// TwinCAT 3 PLC project PLC1
// ProgramVersion: 3.1.4026.19
// CompilerDefines: VISU_USEPROPERTYINFO
// libraries:
//   SimplePackML, * (Beckhoff Automation Poland)
//   Tc2_BABasic, * (Beckhoff Automation GmbH)
//   Tc2_Standard, * (Beckhoff Automation GmbH)
//   Tc2_System, * (Beckhoff Automation GmbH)
//   Tc2_Utilities, * (Beckhoff Automation GmbH)
//   Tc3_EventLogger, * (Beckhoff Automation GmbH)
//   Tc3_PackML_V2, * (Beckhoff Automation GmbH)
// project tree:
//   / ClassDiagram.TcCD (not stored), ClassDiagram_1.TcCD (not stored), GlobalTextList.TcGTLO, PlcTask.TcTTO, Visualization Manager.TcVMO (not stored)
//   POUs/Devices/ Relay.TcPOU, TemperatureSensor.TcPOU
//   POUs/ IncrementVar.TcPOU, IncrementVarInst.TcPOU, MAIN.TcPOU, TestFbInit.TcPOU, Testowy.TcPOU, Testowy2.TcPOU, Testowy3.TcPOU
//   POUs/PackML/ Machine.TcPOU, P_PackML.TcPOU
//   POUs/ZadanieOOP/Devices/ AnalogLedDisplay010.TcPOU, ButtonNO.TcPOU, ButtonNC.TcPOU, Potentiometer.TcPOU
//   POUs/ZadanieOOP/Interfaces/ I_Button.TcIO, I_LimitedStringBuilder.TcIO, I_StringBuilder.TcIO, StringBuilder.TcPOU
//   POUs/ZadanieOOP/Modules/ PumpController.TcPOU, PumpControllerWithLogger.TcPOU, SignalTower.TcPOU, VolumePump.TcPOU
//   POUs/ZadanieOOP/ P_Machine.TcPOU
//   POUs/Zadanie/ FB_JuicePumpSimulator.TcPOU, GVL_IO.TcGVL (excluded from build), P_JuicePump.TcPOU
//   VISUs/ Visualization.TcVIS
// real-time tasks:
//   TASK PlcTask: cycle T#10ms, priority 20, ADS port 350
// I/O:
//   DEVICE Device 1 (EtherCAT), AmsNetId 0.0.0.0.2.1
//     Term 1 (EK1200) [EK1200-5000 EtherCAT Power supply (2A E-Bus)]
//       Term 2 (EL1004) [EL1004 4Ch. Dig. Input 24V, 3ms]
//       Term 3 (EL2008)
//       Term 4 (EL3064) [EL3064 4Ch. Ana. Input 0-10V]
//       Term 5 (EL4008) [EL4008 8Ch. Ana. Output 0-10V, 12bit]
//       Term 6 (EL6910) [EL6910, TwinSAFE PLC]
//       Term 7 (EL6070) [EL6070 1Ch. Licensing-Terminal]
//       Term 8 (EL1904) [EL1904, 4 Ch. Safety Input 24V, TwinSAFE]
//         modules: Module 1 (FSOES)
//       Term 9 (EL2904) [EL2904, 4 Ch. Safety Output 24V, 0.5A, TwinSAFE]
//         modules: Module 1 (FSOES), Module 2 (DO)
//       Term 10 (EL1018) [EL1018 8Ch. Dig. Input 24V, 10µs]
//       Term 11 (EL3214-0090) [EL3214-0090 4Ch. Ana. Input PT100 (RTD), TwinSAFE SC]
//       Term 12 (EL2024) [EL2024 4Ch. Dig. Output 24V, 2A]
//       Term 13 (EK1110) [EK1110 EtherCAT extension]
// variable links:
//   (this object) <-> Device 1 (EtherCAT)/Term 1 (EK1200)/Term 11 (EL3214-0090)
//     PlcTask Inputs/MAIN.tempSensor.stInputData.MDP5001_320_Input/MDP5001_320_Status <-> RTD Inputs Channel 1/Status
//     PlcTask Inputs/MAIN.tempSensor.stInputData.MDP5001_320_Input/MDP5001_320_Value <-> RTD Inputs Channel 1/Value
//   (this object) <-> Device 1 (EtherCAT)/Term 1 (EK1200)/Term 2 (EL1004)
//     PlcTask Inputs/MAIN.testButton.bInput <-> Channel 2/Input
//     PlcTask Inputs/P_Machine.requestButton.bInput <-> Channel 3/Input
//     PlcTask Inputs/P_Machine.startButton.bInput <-> Channel 1/Input
//   (this object) <-> Device 1 (EtherCAT)/Term 1 (EK1200)/Term 3 (EL2008)
//     PlcTask Outputs/P_Machine.appleJuiceContoller.volumePump.pump.bOutput <-> Channel 3/Output
//     PlcTask Outputs/P_Machine.signalTower.lightGreen.bOutput <-> Channel 1/Output
//     PlcTask Outputs/P_Machine.signalTower.lightRed.bOutput <-> Channel 2/Output
//   (this object) <-> Device 1 (EtherCAT)/Term 1 (EK1200)/Term 4 (EL3064)
//     PlcTask Inputs/P_Machine.appleJuiceContoller.juiceSetter.nInput <-> AI Standard Channel 1/Value
//     PlcTask Inputs/P_Machine.orangeJuiceContoller.juiceSetter.nInput <-> AI Standard Channel 2/Value
//   (this object) <-> Device 1 (EtherCAT)/Term 1 (EK1200)/Term 5 (EL4008)
//     PlcTask Outputs/P_Machine.appleJuiceContoller.ledDisplay.nOutput <-> AO Outputs Channel 1/Analog output
//     PlcTask Outputs/P_Machine.orangeJuiceContoller.ledDisplay.nOutput <-> AO Outputs Channel 2/Analog output

CONFIGURATION PLC1
    RESOURCE PLC ON TwinCAT3
        TASK PlcTask(INTERVAL := T#10ms, PRIORITY := 20);
        PROGRAM MAIN WITH PlcTask : MAIN;
    END_RESOURCE
END_CONFIGURATION

// ---- POUs/Zadanie/GVL_IO.TcGVL
{attribute 'qualified_only'}
VAR_GLOBAL
	//wejscia
	bStart			AT%I*	: BOOL;
	bRequest		AT%I*	: BOOL;
	nJuiceSetter	AT%I*	: INT;
	//wyścia
	bLightSignal1	AT%Q*	: BOOL;
	bLightSignal2	AT%Q*	: BOOL;
	nLedDisplay		AT%Q*	: INT;
	bPump			AT%Q*	: BOOL;
END_VAR

// ---- POUs/ZadanieOOP/Interfaces/I_Button.TcIO
INTERFACE I_Button

PROPERTY IsPressed : BOOL
GET
END_GET
END_PROPERTY

PROPERTY IsReleased : BOOL
GET
END_GET
END_PROPERTY

PROPERTY RisingTrigger : BOOL
GET
END_GET
END_PROPERTY

END_INTERFACE

// ---- POUs/ZadanieOOP/Interfaces/I_LimitedStringBuilder.TcIO
INTERFACE I_LimitedStringBuilder

METHOD Append : I_StringBuilder
VAR_INPUT
	sText	: T_MaxString;
END_VAR
END_METHOD

METHOD Reset : I_LimitedStringBuilder
VAR_INPUT
END_VAR
END_METHOD

METHOD ToString : T_MaxString
VAR_INPUT
END_VAR
END_METHOD

END_INTERFACE

// ---- POUs/ZadanieOOP/Interfaces/I_StringBuilder.TcIO
INTERFACE I_StringBuilder

METHOD Append : I_StringBuilder
VAR_INPUT
	sText	: T_MaxString;
END_VAR
END_METHOD

METHOD Reset : I_LimitedStringBuilder
VAR_INPUT
END_VAR
END_METHOD

METHOD ToLowerCase : I_StringBuilder
VAR_INPUT
END_VAR
END_METHOD

METHOD ToString : T_MaxString
VAR_INPUT
END_VAR
END_METHOD

METHOD ToUpperCase : I_StringBuilder
VAR_INPUT
END_VAR
END_METHOD

END_INTERFACE

// ---- POUs/MAIN.TcPOU
PROGRAM MAIN
VAR
	nState		: UINT;
	motorRelay	: Relay;
	incVar		: IncrementVar;
	incVarInst	: IncrementVarInst;
	bTest		: BOOL;
	nVal1		: INT;
	nVal2		: INT;
	tempSensor	: TemperatureSensor;
	temperature	: REAL;
	offset		: REAL;
	
	testButton	: ButtonNC;
	testTrigger	: BOOL;
	
	testFbInit	: TestFbInit(wartosc := 7);
	
	pInt		: REFERENCE TO INT;
	nInt		: INT;
	nInt2		: INT;
	
	itfButton	: I_Button;
	buttonNo	: ButtonNO;
	buttonNc	: ButtonNC;
	bIsPressed	: BOOL;
	
	sTekst		: STRING;
	nNrAlarmu	: INT := 7;
	alarm 		: StringBuilder;
END_VAR

motorRelay.Cyclic();

CASE nState OF
	
	0:
		;
		
	10:
		IF motorRelay.SwitchOn() THEN
			nState := 0;
		END_IF
		
	20:
		IF motorRelay.SwitchOff() THEN
			nState := 0;
		END_IF
		
	30:
		IF motorRelay.Pulse(T#5S) THEN
			nState := 0;
		END_IF
		
	40:
		IF motorRelay.PulseAcyclic(T#5S) THEN
			nState := 0;
		END_IF
		
END_CASE

IF bTest THEN
	bTest := FALSE;
	nVal1 := incVar.Increment();
	nVal2 := incVarInst.Increment();
END_IF

tempSensor.OffsetInCelsius := -25;
temperature := tempSensor.InCelsius;
offset := tempSensor.OffsetInCelsius;

// P_JuicePump();
P_Machine();

IF testButton.RisingTrigger THEN
	testTrigger := TRUE;
END_IF

pInt REF= nInt2;

IF __ISVALIDREF(pInt) THEN
	nInt := pInt;
END_IF

itfButton := buttonNc;

IF itfButton <> 0 AND_THEN itfButton.IsPressed THEN
	bIsPressed := TRUE;
END_IF

// sTekst := alarm.Reset()
// 			.Append('Alarm nr: ')
// 			.Append(TO_STRING(nNrAlarmu))
// 			.Append(' Temperatura zbyt wysoka')
// 			.ToString();

P_PackML();

END_PROGRAM

// ---- POUs/Devices/Relay.TcPOU
FUNCTION_BLOCK Relay
VAR
	bOutput	AT%Q*	: BOOL;
	tonPulse		: TON;
	tonPulseAcyclic	: TON;
END_VAR

// tonPulseAcyclic();
// 
// IF tonPulseAcyclic.Q THEN
// 	SwitchOff();
// 	tonPulseAcyclic(IN := FALSE);
// END_IF

METHOD Cyclic
VAR_INPUT
END_VAR
tonPulseAcyclic();

IF tonPulseAcyclic.Q THEN
	SwitchOff();
	tonPulseAcyclic(IN := FALSE);
END_IF
END_METHOD

METHOD Pulse : BOOL
VAR_INPUT
	tPulseTime	: TIME;
END_VAR
tonPulse(IN := TRUE, PT:= tPulseTime);

IF NOT tonPulse.Q THEN
	SwitchOn();
ELSIF tonPulse.Q THEN
	SwitchOff();
	tonPulse(IN := FALSE);
	Pulse := TRUE;
END_IF
END_METHOD

METHOD PulseAcyclic : BOOL
VAR_INPUT
	tPulseTime	: TIME;
END_VAR
SwitchOn();
tonPulseAcyclic.IN := TRUE;
tonPulseAcyclic.PT := tPulseTime;

PulseAcyclic := TRUE;
END_METHOD

PROPERTY State : BOOL
GET
State := bOutput;
END_GET
END_PROPERTY

METHOD SwitchOff : BOOL
VAR_INPUT
END_VAR
bOutput := FALSE;

SwitchOff := TRUE;
END_METHOD

METHOD SwitchOn : BOOL
VAR_INPUT
END_VAR
bOutput := TRUE;

SwitchOn := TRUE;
END_METHOD

END_FUNCTION_BLOCK

// ---- POUs/IncrementVar.TcPOU
FUNCTION_BLOCK IncrementVar
VAR
END_VAR

METHOD Increment : INT
VAR
	nValue	: INT := 5;
END_VAR
nValue := nValue + 1;
Increment := nValue;
END_METHOD

END_FUNCTION_BLOCK

// ---- POUs/IncrementVarInst.TcPOU
FUNCTION_BLOCK IncrementVarInst
VAR
END_VAR

METHOD Increment : INT
VAR_INST
	nValue	: INT := 5;
END_VAR
nValue := nValue + 1;
Increment := nValue;
END_METHOD

END_FUNCTION_BLOCK

// ---- POUs/Devices/TemperatureSensor.TcPOU
FUNCTION_BLOCK TemperatureSensor
VAR
	stInputData			: MDP5001_320_A369A904;
	fOffsetInCelsius	: REAL;
END_VAR

{attribute 'monitoring' := 'call'}
PROPERTY Error : BOOL
GET
Error := stInputData.MDP5001_320_Input.MDP5001_320_Status.Error;
END_GET
END_PROPERTY

{attribute 'monitoring' := 'call'}
PROPERTY InCelsius : REAL
GET
InCelsius := (stInputData.MDP5001_320_Input.MDP5001_320_Value / 10.0) + fOffsetInCelsius;
END_GET
END_PROPERTY

{attribute 'monitoring' := 'call'}
PROPERTY InFarenheit : REAL
GET
InFarenheit := C_TO_F ( fX := InCelsius );
END_GET
END_PROPERTY

{attribute 'monitoring' := 'call'}
PROPERTY InKelvin : REAL
GET
InKelvin := C_TO_K ( fX := InCelsius );
END_GET
END_PROPERTY

{attribute 'monitoring' := 'call'}
PROPERTY InReaumur : REAL
GET
InReaumur := C_TO_R ( fX := InCelsius );
END_GET
END_PROPERTY

{attribute 'monitoring' := 'call'}
PROPERTY OffsetInCelsius : REAL
GET
OffsetInCelsius := fOffsetInCelsius;
END_GET
SET
fOffsetInCelsius := OffsetInCelsius;
END_SET
END_PROPERTY

{attribute 'monitoring' := 'call'}
PROPERTY Overrange : BOOL
GET
Overrange := stInputData.MDP5001_320_Input.MDP5001_320_Status.Overrange;
END_GET
END_PROPERTY

{attribute 'monitoring' := 'call'}
PROPERTY Underrange : BOOL
GET
Underrange := stInputData.MDP5001_320_Input.MDP5001_320_Status.Underrange;
END_GET
END_PROPERTY

END_FUNCTION_BLOCK

// ---- POUs/ZadanieOOP/Devices/ButtonNC.TcPOU
FUNCTION_BLOCK ButtonNC IMPLEMENTS I_Button
VAR
	bInput	AT%I*	: BOOL;
	rtInput			: R_TRIG;
END_VAR

PROPERTY IsPressed : BOOL
GET
IsPressed := NOT bInput;
END_GET
END_PROPERTY

PROPERTY IsReleased : BOOL
GET
IsReleased := NOT IsPressed;
END_GET
END_PROPERTY

PROPERTY RisingTrigger : BOOL
GET
rtInput(CLK := IsPressed);

RisingTrigger := rtInput.Q;
END_GET
END_PROPERTY

END_FUNCTION_BLOCK

// ---- POUs/TestFbInit.TcPOU
FUNCTION_BLOCK TestFbInit
VAR
	nValue	: INT := 5;
END_VAR

//FB_Init is always available implicitly and it is used primarily for initialization.
//The return value is not evaluated. For a specific influence, you can also declare the
//methods explicitly and provide additional code there with the standard initialization
//code. You can evaluate the return value.
METHOD FB_Init: BOOL
VAR_INPUT
    bInitRetains: BOOL; // TRUE: the retain variables are initialized (reset warm / reset cold)
    bInCopyCode: BOOL;  // TRUE: the instance will be copied to the copy code afterward (online change)
	wartosc		: INT;   
END_VAR
nValue := wartosc;
END_METHOD

END_FUNCTION_BLOCK

// ---- POUs/ZadanieOOP/Devices/ButtonNO.TcPOU
FUNCTION_BLOCK ButtonNO IMPLEMENTS I_Button
VAR
	bInput	AT%I*	: BOOL;
	rtInput			: R_TRIG;
END_VAR

PROPERTY IsPressed : BOOL
GET
IsPressed := bInput;
END_GET
END_PROPERTY

PROPERTY IsReleased : BOOL
GET
IsReleased := NOT IsPressed;
END_GET
END_PROPERTY

PROPERTY RisingTrigger : BOOL
GET
rtInput(CLK := IsPressed);

RisingTrigger := rtInput.Q;
END_GET
END_PROPERTY

END_FUNCTION_BLOCK

// ---- POUs/ZadanieOOP/Interfaces/StringBuilder.TcPOU
FUNCTION_BLOCK StringBuilder IMPLEMENTS I_LimitedStringBuilder, I_StringBuilder
VAR
	sBuiltString	: T_MaxString;
END_VAR

METHOD Append : I_StringBuilder
VAR_INPUT
	sText	: T_MaxString;
END_VAR
sBuiltString := CONCAT(sBuiltString, sText);

Append := THIS^;
END_METHOD

METHOD Reset : I_LimitedStringBuilder
sBuiltString := '';

Reset := THIS^;
END_METHOD

{warning 'Add method implementation '}
METHOD ToLowerCase : I_StringBuilder
END_METHOD

METHOD ToString : T_MaxString
ToString := sBuiltString;
END_METHOD

{warning 'Add method implementation '}
METHOD ToUpperCase : I_StringBuilder
END_METHOD

END_FUNCTION_BLOCK

// ---- POUs/ZadanieOOP/P_Machine.TcPOU
PROGRAM P_Machine
VAR
	startButton			: ButtonNO;
	requestButton		: ButtonNO;
	appleJuiceContoller	: PumpControllerWithLogger(requestButton, 0, 10_000);
	orangeJuiceContoller: PumpControllerWithLogger(requestButton, 0, 5_000);
	signalTower			: SignalTower;
END_VAR

appleJuiceContoller();
orangeJuiceContoller();

IF startButton.RisingTrigger THEN
	appleJuiceContoller.Enable();
	orangeJuiceContoller.Enable();
END_IF

IF appleJuiceContoller.IsDisabled THEN
	signalTower.SwitchOffGreen();
	signalTower.SwitchOffRed();
ELSIF appleJuiceContoller.IsEnabled THEN
	signalTower.SwitchOnGreen();
	signalTower.SwitchOffRed();
ELSIF appleJuiceContoller.IsPumping THEN
	signalTower.SwitchOnGreen();
	signalTower.SwitchOnRed();
ELSIF appleJuiceContoller.IsPumpingComplete THEN
	signalTower.SwitchOnGreen();
	signalTower.SwitchOffRed();
END_IF

END_PROGRAM

// ---- POUs/ZadanieOOP/Modules/PumpControllerWithLogger.TcPOU
FUNCTION_BLOCK PumpControllerWithLogger EXTENDS PumpController
VAR
	stringBuilder	: StringBuilder;
	logDataTrigger	: R_TRIG;
END_VAR
VAR_STAT
	nCycles			: UINT;
END_VAR

SUPER^();

LogToAds();

METHOD PRIVATE LogToAds : BOOL
VAR_INPUT
END_VAR
logDataTrigger(CLK := IsPumpingComplete);

IF logDataTrigger.Q THEN
	nCycles := nCycles + 1;
	
	stringBuilder.Reset()
		.Append('Lacznie wykonano: ')
		.Append(TO_STRING(nCycles))
		.Append(' cykli');
		
	ADSLOGSTR( msgCtrlMask := ADSLOG_MSGTYPE_LOG, msgFmtStr := stringBuilder.ToString(), strArg := '' );
END_IF
END_METHOD

END_FUNCTION_BLOCK

// ---- POUs/ZadanieOOP/Modules/PumpController.TcPOU
FUNCTION_BLOCK PumpController
VAR
	volumePump					: VolumePump;
	eState						: ( DISABLED, ENABLED, PUMPING, PUMPING_COMPLETE );
	requestButton				: I_Button;
	juiceSetter					: Potentiometer;
	ledDisplay					: AnalogLedDisplay010;
	fJuiceSetpointInMililiters	: LREAL;
	fMinSetRangeInMililiters	: LREAL;
	fMaxSetRangeInMililiters	: LREAL;
END_VAR

volumePump();

CASE eState OF
	
	DISABLED:
		;
		
	ENABLED:
		ledDisplay.SetValue(juiceSetter.ActualValue);
		IF requestButton.IsPressed THEN
			fJuiceSetpointInMililiters := F_Scale ( juiceSetter.ActualValue, 0, 32767, fMinSetRangeInMililiters, fMaxSetRangeInMililiters );
			eState := PUMPING;
		END_IF
		
	PUMPING:
		ledDisplay.SetValue( TO_INT (F_Scale ( fJuiceSetpointInMililiters - volumePump.PumpedJuiceInMililiters, fMinSetRangeInMililiters, fMaxSetRangeInMililiters, 0, 32767 ) ) );
		volumePump.Start();
		IF volumePump.PumpedJuiceInMililiters >= fJuiceSetpointInMililiters THEN
			volumePump.Reset();
			eState := PUMPING_COMPLETE;
		END_IF
		
	PUMPING_COMPLETE:
		;
		
END_CASE

METHOD Disable : BOOL
VAR_INPUT
END_VAR
eState := DISABLED;
END_METHOD

METHOD Enable : BOOL
VAR_INPUT
END_VAR
eState := ENABLED;
END_METHOD

//FB_Init is always available implicitly and it is used primarily for initialization.
//The return value is not evaluated. For a specific influence, you can also declare the
//methods explicitly and provide additional code there with the standard initialization
//code. You can evaluate the return value.
METHOD FB_Init: BOOL
VAR_INPUT
    bInitRetains: BOOL; // TRUE: the retain variables are initialized (reset warm / reset cold)
    bInCopyCode: BOOL;  // TRUE: the instance will be copied to the copy code afterward (online change)   
	requestButton				: I_Button;
	fMinSetRangeInMililiters	: LREAL;
	fMaxSetRangeInMililiters	: LREAL;
END_VAR
THIS^.requestButton := requestButton;
THIS^.fMinSetRangeInMililiters := LIMIT(0, fMinSetRangeInMililiters, 10_000);
THIS^.fMaxSetRangeInMililiters := LIMIT(0, fMaxSetRangeInMililiters, 10_000);
END_METHOD

PROPERTY IsDisabled : BOOL
GET
IsDisabled := eState = DISABLED;
END_GET
END_PROPERTY

PROPERTY IsEnabled : BOOL
GET
IsEnabled := eState = ENABLED;
END_GET
END_PROPERTY

PROPERTY IsPumping : BOOL
GET
IsPumping := eState = PUMPING;
END_GET
END_PROPERTY

PROPERTY IsPumpingComplete : BOOL
GET
IsPumpingComplete := eState = PUMPING_COMPLETE;
END_GET
END_PROPERTY

END_FUNCTION_BLOCK

// ---- POUs/ZadanieOOP/Modules/VolumePump.TcPOU
FUNCTION_BLOCK VolumePump
VAR
	pump						: Relay;
	eState						: ( RESET, START );
	fPumpedJuiceInMililiters	: REAL;
END_VAR

CASE eState OF
	
	RESET:
		pump.SwitchOff();
		fPumpedJuiceInMililiters := 0;
		
	START:
		pump.SwitchOn();
		fPumpedJuiceInMililiters := fPumpedJuiceInMililiters + 10;
		
END_CASE

PROPERTY IsPumping : BOOL
GET
IsPumping := pump.State;
END_GET
END_PROPERTY

PROPERTY PumpedJuiceInMililiters : REAL
GET
PumpedJuiceInMililiters := fPumpedJuiceInMililiters;
END_GET
END_PROPERTY

METHOD Reset : BOOL
VAR_INPUT
END_VAR
eState := RESET;
END_METHOD

METHOD Start : BOOL
VAR_INPUT
END_VAR
eState := START;
END_METHOD

END_FUNCTION_BLOCK

// ---- POUs/ZadanieOOP/Devices/Potentiometer.TcPOU
FUNCTION_BLOCK Potentiometer
VAR
	nInput	AT%I*	: INT;
END_VAR

PROPERTY ActualValue : INT
GET
ActualValue := nInput;
END_GET
END_PROPERTY

PROPERTY ActualValuePercent : LREAL
GET
ActualValuePercent := F_Scale ( nInput, 0, 32767, 0, 100 );
END_GET
END_PROPERTY

END_FUNCTION_BLOCK

// ---- POUs/ZadanieOOP/Devices/AnalogLedDisplay010.TcPOU
FUNCTION_BLOCK AnalogLedDisplay010
VAR
	nOutput	AT%Q*	: INT;
END_VAR

PROPERTY DisplayedValue : LREAL
GET
DisplayedValue := F_Scale ( nOutput, 0, 32767, 0, 10 );
END_GET
END_PROPERTY

METHOD SetValue : BOOL
VAR_INPUT
	nValue	: INT;
END_VAR
nOutput := nValue;

SetValue := TRUE;
END_METHOD

END_FUNCTION_BLOCK

// ---- POUs/ZadanieOOP/Modules/SignalTower.TcPOU
FUNCTION_BLOCK SignalTower
VAR
	lightGreen	: Relay;
	lightRed	: Relay;
END_VAR

PROPERTY GreenLightState : BOOL
GET
GreenLightState := lightGreen.State;
END_GET
END_PROPERTY

PROPERTY RedLightState : BOOL
GET
RedLightState := lightRed.State;
END_GET
END_PROPERTY

METHOD SwitchOffGreen : BOOL
VAR_INPUT
END_VAR
lightGreen.SwitchOff();
END_METHOD

METHOD SwitchOffRed : BOOL
VAR_INPUT
END_VAR
lightRed.SwitchOff();
END_METHOD

METHOD SwitchOnGreen : BOOL
VAR_INPUT
END_VAR
lightGreen.SwitchOn();
END_METHOD

METHOD SwitchOnRed : BOOL
VAR_INPUT
END_VAR
lightRed.SwitchOn();
END_METHOD

END_FUNCTION_BLOCK

// ---- POUs/PackML/P_PackML.TcPOU
PROGRAM P_PackML
VAR
	machine1	: Machine;
	eModeCommand: E_PMLProtectedUnitMode;
	eCommand	: E_PMLCommand;
END_VAR

machine1(
	eModeCommand	:= eModeCommand, 
	eCommand		:= eCommand, 
	eMode			=> , 
	eState			=> , 
	bUndefinedDone	=> , 
	bInvalidModeCommandOut=> , 
	bChangeIntoProduction=> );

END_PROGRAM

// ---- POUs/PackML/Machine.TcPOU
FUNCTION_BLOCK Machine EXTENDS FB_Generic
VAR
END_VAR

SUPER^();

METHOD M_Aborting
VAR_INST
	bTest	: BOOL;
END_VAR
IF bTest THEN
	bTest := FALSE;
	M_StateComplete();
END_IF
END_METHOD

METHOD M_Execute
VAR_INST
	bTest	: BOOL;
END_VAR
IF bTest THEN
	bTest := FALSE;
	M_StateComplete();
END_IF
END_METHOD

METHOD M_StateComplete
SUPER^.M_StateComplete();
END_METHOD

END_FUNCTION_BLOCK

// ---- POUs/Testowy.TcPOU
FUNCTION_BLOCK Testowy
VAR
END_VAR

END_FUNCTION_BLOCK

// ---- POUs/Testowy2.TcPOU
FUNCTION_BLOCK Testowy2
VAR
	bTest: BOOL;
END_VAR

END_FUNCTION_BLOCK

// ---- POUs/Testowy3.TcPOU
FUNCTION_BLOCK Testowy3
VAR
	bTest3: BOOL;
END_VAR

END_FUNCTION_BLOCK

// ---- POUs/Zadanie/FB_JuicePumpSimulator.TcPOU
FUNCTION_BLOCK FB_JuicePumpSimulator
VAR_INPUT
	bStart						: BOOL;
	bReset						: BOOL;
END_VAR
VAR_OUTPUT
	fPumpedJuiceInMililiters	: REAL;
END_VAR
VAR
	rtReset						: R_TRIG;
END_VAR

rtReset( CLK := bReset );
IF rtReset.Q THEN
	fPumpedJuiceInMililiters := 0;
END_IF

IF bStart THEN
	fPumpedJuiceInMililiters := fPumpedJuiceInMililiters + 10;		// 1kg / s
END_IF

END_FUNCTION_BLOCK

// ---- POUs/Zadanie/P_JuicePump.TcPOU
PROGRAM P_JuicePump
VAR
	eState						: ( DISABLED, ENABLED, PUMPING );
	fbPumpSimulator				: FB_JuicePumpSimulator;
	rtStartButton				: R_TRIG;
	ftStartButton				: F_TRIG;
	fJuiceSetpointInMililiters	: LREAL;
END_VAR

fbPumpSimulator( bStart := GVL_IO.bPump );
ftStartButton( CLK := GVL_IO.bStart );
IF ftStartButton.Q THEN
	fbPumpSimulator( bReset := TRUE );
	fbPumpSimulator( bReset := FALSE );
END_IF

CASE eState OF
	
	DISABLED:
		rtStartButton(CLK := GVL_IO.bStart);
		IF rtStartButton.Q THEN
			eState := ENABLED;
		END_IF
		
	ENABLED:
		GVL_IO.bLightSignal1 := TRUE;
		GVL_IO.nLedDisplay := GVL_IO.nJuiceSetter;
		IF GVL_IO.bRequest THEN
			fJuiceSetpointInMililiters := F_Scale ( GVL_IO.nJuiceSetter, 0, 32767, 0, 10_000 );
			eState := PUMPING;
		END_IF
		
	PUMPING:
		GVL_IO.nLedDisplay := TO_INT (F_Scale ( fJuiceSetpointInMililiters - fbPumpSimulator.fPumpedJuiceInMililiters, 0, 10_000, 0, 32767 ) );
		GVL_IO.bLightSignal2 := TRUE;
		GVL_IO.bPump := TRUE;
		IF fbPumpSimulator.fPumpedJuiceInMililiters >= fJuiceSetpointInMililiters THEN
			GVL_IO.bLightSignal1 := FALSE;
			GVL_IO.bLightSignal2 := FALSE;
			GVL_IO.bPump := FALSE;
			eState := DISABLED;
		END_IF
		
END_CASE

END_PROGRAM

// ---- VISUs/Visualization.TcVIS
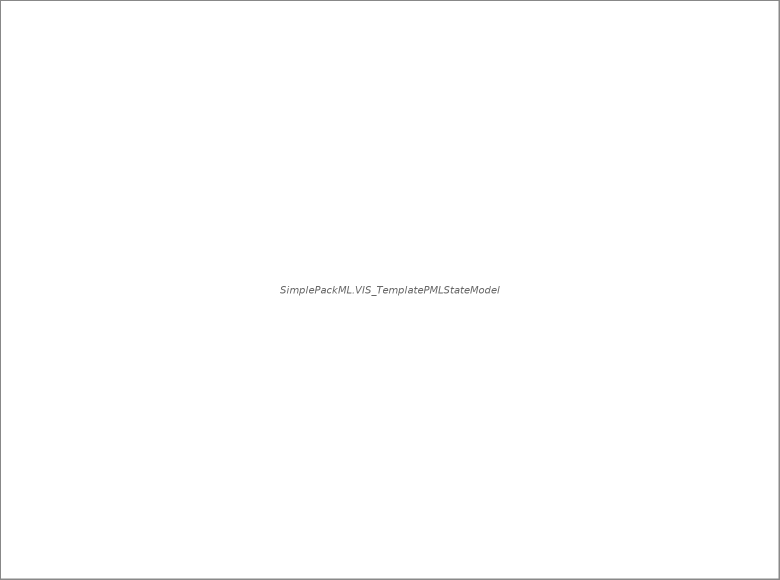
VISUALIZATION Visualization  // 780x580
    Frame (0,0 780x580)
        shows SimplePackML.VIS_TemplatePMLStateModel(ePMLUnitMode := P_PackML.machine1.eMode, ePMLState := P_PackML.machine1.eState)
END_VISUALIZATION
